TYPE (* A Template for a Data Type *)
  (* Version 1.0, 2022-06-27, AK115394 *)
  structtype : STRUCT
    VAR1 : BOOL;
    VAR2 : BOOL;
    VAR3 : BOOL;
    VAR4 : BOOL;
  END_STRUCT;
END_TYPE
